// Mitsubishi GX Works2 project: b12   PLC: Q02/Q02H

PROGRAM MAIN
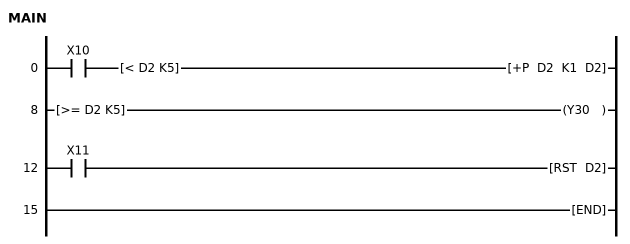
0     LD      X10
      AND<    D2 K5
      +P      D2 K1 D2
8     LD>=    D2 K5
      OUT     Y30
12    LD      X11
      RST     D2
15    END
END_PROGRAM

PROGRAM MAIN1
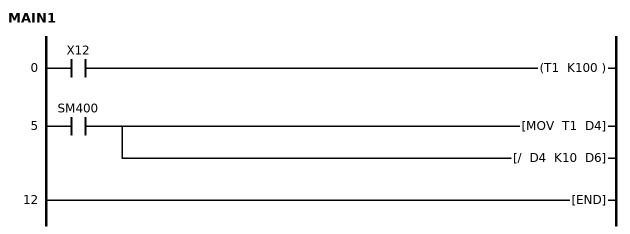
0     LD      X12
      OUT     T1 K100
5     LD      SM400
      MOV     T1 D4
      /       D4 K10 D6
12    END
END_PROGRAM
